// TIA Portal V19 export
DATA_BLOCK "PumpValve"   // DB17
// stored: InstanceOfName Valve_Type, InstanceOfType FB
"Valve_Type"
   // VAR_INPUT
   //    Auto_OPN : Bool;
   //    ManOpen : Bool;
   //    FeedbackFitted : Bool;
   //    FeedbackTime : Time;
   //    Close_Feedback : Bool;
   //    Open_Feedback : Bool;
   //    Global_Reset : Bool;
   //    Simulation : Bool;
   // END_VAR
   // VAR_OUTPUT
   //    "Valve Open" : Bool;
   //    "HMI Valve Open" : Bool;
   //    "HMI Valve Close" : Bool;
   //    "Valve Open Fault" : Bool;
   //    "Valve Close Fault" : Bool;
   // END_VAR
   // VAR_IN_OUT
   //    "Valve Angle" : Real;
   // END_VAR
   // VAR
   //    IEC_Timer_0_Instance { S7_SetPoint := 'True'} : TON_TIME;
   //    IEC_Timer_0_Instance_1 { S7_SetPoint := 'True'} : TON_TIME;
   //    "trig 1" : Bool;
   //    "trig 2" : Bool;
   // END_VAR
BEGIN
END_DATA_BLOCK
